// Mitsubishi GX Works2 project: IELET2103_Datalab4   PLC: FX2N/FX2NC
// IELET2103_Datalab4

// global labels: Global1
VAR_GLOBAL
  BrusInn : BOOL;
  SjokoladeInn : BOOL;
  BrusUt : BOOL;
  SjokoladeUt : BOOL;
  VarselBrus : BOOL;
  VarselSjokolade : BOOL;
  AlarmBrus : BOOL;
  AlarmSjokolade : BOOL;
  TomtForVare : BOOL;
  AntallBrus : WORD;
  AntallSjokolade : WORD;
END_VAR

// task Task_01 (event TRUE, interval 0, priority 31): Oppgave1

PROGRAM Oppgave1
(* structured ladder/FBD written out as ST: instructions are called as NAME(EN, inputs, outputs); _pN, _eN, _tN stand for wires *)
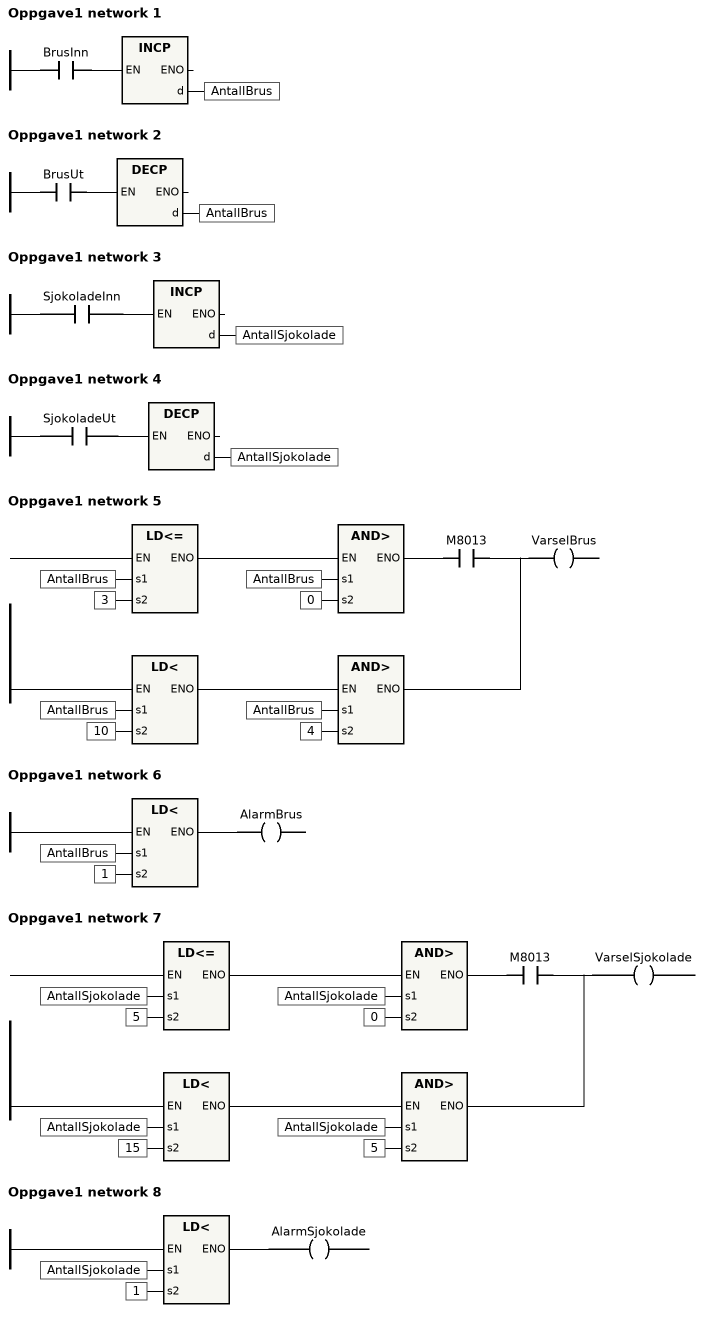
(* network 1 *)
INCP(BrusInn, AntallBrus);
(* network 2 *)
DECP(BrusUt, AntallBrus);
(* network 3 *)
INCP(SjokoladeInn, AntallSjokolade);
(* network 4 *)
DECP(SjokoladeUt, AntallSjokolade);
(* network 5 *)
_e1 := LD<=(TRUE, AntallBrus, 3);
_e2 := AND>(_e1, AntallBrus, 0);
_e3 := LD<(TRUE, AntallBrus, 10);
_e4 := AND>(_e3, AntallBrus, 4);
VarselBrus := (_e2 AND M8013) OR _e4;
(* network 6 *)
_e1 := LD<(TRUE, AntallBrus, 1);
AlarmBrus := _e1;
(* network 7 *)
_e1 := LD<=(TRUE, AntallSjokolade, 5);
_e2 := AND>(_e1, AntallSjokolade, 0);
_e3 := LD<(TRUE, AntallSjokolade, 15);
_e4 := AND>(_e3, AntallSjokolade, 5);
VarselSjokolade := (_e2 AND M8013) OR _e4;
(* network 8 *)
_e1 := LD<(TRUE, AntallSjokolade, 1);
AlarmSjokolade := _e1;
END_PROGRAM

PROGRAM Oppgave1c
(* structured ladder/FBD written out as ST: instructions are called as NAME(EN, inputs, outputs); _pN, _eN, _tN stand for wires *)
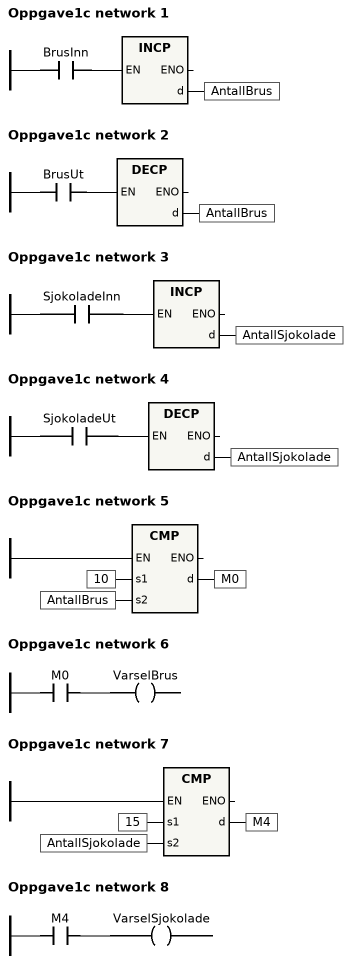
(* network 1 *)
INCP(BrusInn, AntallBrus);
(* network 2 *)
DECP(BrusUt, AntallBrus);
(* network 3 *)
INCP(SjokoladeInn, AntallSjokolade);
(* network 4 *)
DECP(SjokoladeUt, AntallSjokolade);
(* network 5 *)
CMP(TRUE, 10, AntallBrus, M0);
(* network 6 *)
VarselBrus := M0;
(* network 7 *)
CMP(TRUE, 15, AntallSjokolade, M4);
(* network 8 *)
VarselSjokolade := M4;
END_PROGRAM
